// TIA Portal V16 export
// export: Created 2021-11-12T13:31:27.948898Z, ExportSetting WithDefaults, DisplayName Totally Integrated Automation Portal, DisplayVersion V16 Update 3, DisplayName TIA Portal Version Control Interface, DisplayVersion V16 Update 2, DisplayName TIA Portal Openness, DisplayVersion V16 Update 3, DisplayName SINAMICS Startdrive Advanced, DisplayVersion V16 Update 5, DisplayName SINAMICS Startdrive G130, G150, S120, S150, SINAMICS MV, S210, DisplayVersion V16 Update 5, DisplayName SINAMICS Startdrive G110M, G120, G120C, G120D, G120P, G115D, DisplayVersion V16 Update 5, DisplayName STEP 7 Professional, DisplayVersion V16 Update 3, DisplayName STEP 7 Safety, DisplayVersion V16, DisplayName WinCC UA Professional, DisplayVersion V16 Update 3
FUNCTION "MTS_UpdateState" : Void   // FC13, LAD
TITLE = Update state
{ S7_Optimized_Access := 'TRUE' }
VERSION : 0.1
// Update state of the position according to material data flags
// stored: AutoNumber true, IsIECCheckEnabled false, SetENOAutomatically false, UDAEnableTagReadback false
   VAR_IN_OUT
      XS_MaterialData : "UDT_MatCard";
   END_VAR
   VAR_TEMP
      TI_State : Int;
   END_VAR
BEGIN

REGION Network 1: Part is not OK
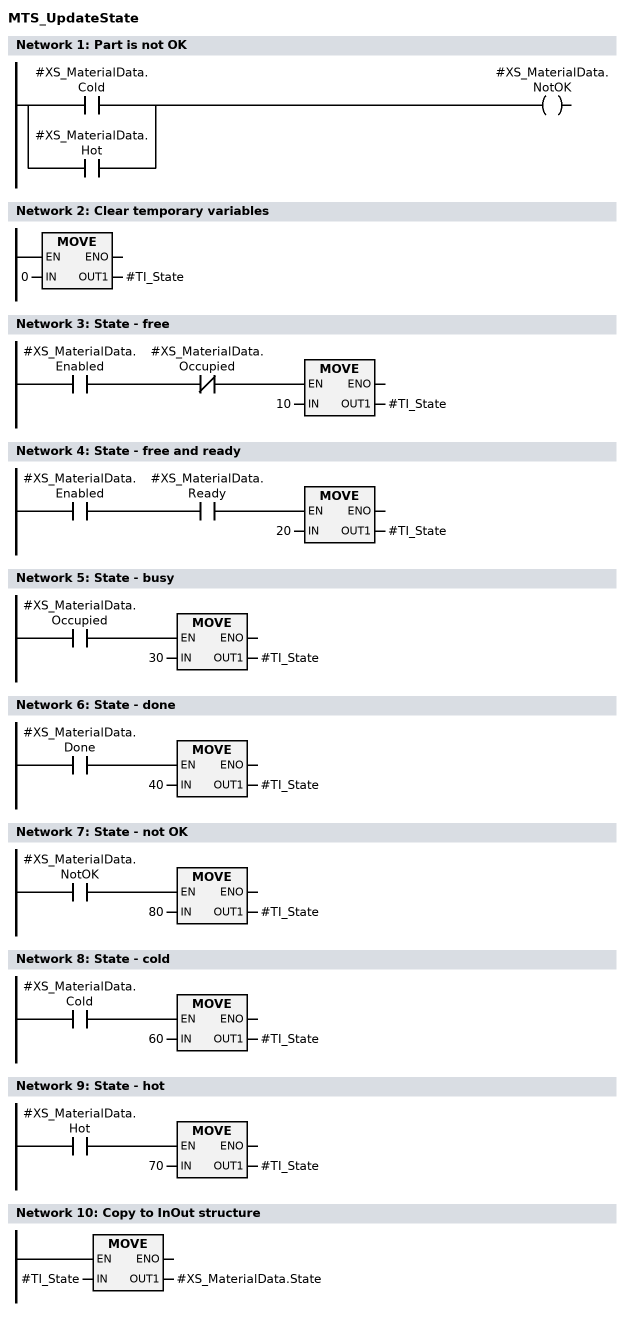
   RUNG wire#powerrail
      Contact( #XS_MaterialData.Cold )
      wire#w1
      Coil( #XS_MaterialData.NotOK )
   END_RUNG
   RUNG wire#powerrail
      Contact( #XS_MaterialData.Hot )
   END_RUNG wire#w1
   // the same network as SCL:
   #XS_MaterialData.NotOK := #XS_MaterialData.Cold OR #XS_MaterialData.Hot;
END_REGION

REGION Network 2: Clear temporary variables
   RUNG wire#powerrail
      Move(in := 0, out1 => #TI_State)
   END_RUNG
   // the same network as SCL:
   #TI_State := 0;
END_REGION

REGION Network 3: State - free
   RUNG wire#powerrail
      Contact( #XS_MaterialData.Enabled )
      I_Contact( #XS_MaterialData.Occupied )
      Move(in := 10, out1 => #TI_State)
   END_RUNG
   // the same network as SCL:
   IF #XS_MaterialData.Enabled AND NOT #XS_MaterialData.Occupied THEN #TI_State := 10; END_IF;
END_REGION

REGION Network 4: State - free and ready
   RUNG wire#powerrail
      Contact( #XS_MaterialData.Enabled )
      Contact( #XS_MaterialData.Ready )
      Move(in := 20, out1 => #TI_State)
   END_RUNG
   // the same network as SCL:
   IF #XS_MaterialData.Enabled AND #XS_MaterialData.Ready THEN #TI_State := 20; END_IF;
END_REGION

REGION Network 5: State - busy
   RUNG wire#powerrail
      Contact( #XS_MaterialData.Occupied )
      Move(in := 30, out1 => #TI_State)
   END_RUNG
   // the same network as SCL:
   IF #XS_MaterialData.Occupied THEN #TI_State := 30; END_IF;
END_REGION

REGION Network 6: State - done
   RUNG wire#powerrail
      Contact( #XS_MaterialData.Done )
      Move(in := 40, out1 => #TI_State)
   END_RUNG
   // the same network as SCL:
   IF #XS_MaterialData.Done THEN #TI_State := 40; END_IF;
END_REGION

REGION Network 7: State - not OK
   RUNG wire#powerrail
      Contact( #XS_MaterialData.NotOK )
      Move(in := 80, out1 => #TI_State)
   END_RUNG
   // the same network as SCL:
   IF #XS_MaterialData.NotOK THEN #TI_State := 80; END_IF;
END_REGION

REGION Network 8: State - cold
   RUNG wire#powerrail
      Contact( #XS_MaterialData.Cold )
      Move(in := 60, out1 => #TI_State)
   END_RUNG
   // the same network as SCL:
   IF #XS_MaterialData.Cold THEN #TI_State := 60; END_IF;
END_REGION

REGION Network 9: State - hot
   RUNG wire#powerrail
      Contact( #XS_MaterialData.Hot )
      Move(in := 70, out1 => #TI_State)
   END_RUNG
   // the same network as SCL:
   IF #XS_MaterialData.Hot THEN #TI_State := 70; END_IF;
END_REGION

REGION Network 10: Copy to InOut structure
   RUNG wire#powerrail
      Move(in := #TI_State, out1 => #XS_MaterialData.State)
   END_RUNG
   // the same network as SCL:
   #XS_MaterialData.State := #TI_State;
END_REGION
END_FUNCTION
